// TIA Portal V19 export
FUNCTION_BLOCK "DelayOnOff"   // FB113, LAD
TITLE = Delay ON-OFF for sensor / DELAY ON/OFF
// stored: MemoryReserve 100, SetENOAutomatically false
   VAR_INPUT
      IN : Bool;
      DelayON : Time;
      DelayOFF : Time;
   END_VAR
   VAR_OUTPUT
      OUT : Bool;
   END_VAR
   VAR
      tonDelayOn : IEC_TIMER;
      tonDelayOff : IEC_TIMER;
   END_VAR
   VAR DB_SPECIFIC
      Result : Bool;
   END_VAR
BEGIN

REGION Network 1: Delay ON-OFF / Main
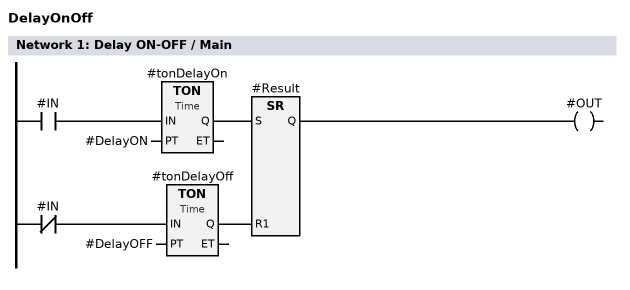
   RUNG wire#powerrail
      Contact( #IN )
      { S7_Templates := "time_type := Time" } #tonDelayOn.TON(pt := #DelayON, et =>)
      S_SR(operand := #Result, r1 := wire#w1)
      Coil( #OUT )
   END_RUNG
   RUNG wire#powerrail
      I_Contact( #IN )
      { S7_Templates := "time_type := Time" } #tonDelayOff.TON(pt := #DelayOFF, et =>)
   END_RUNG wire#w1
   // the same network as SCL:
   #tonDelayOn.TON(IN := #IN, PT := #DelayON);
   #tonDelayOff.TON(IN := NOT #IN, PT := #DelayOFF);
   IF #tonDelayOn.Q THEN
       #Result := TRUE;   // SR flip-flop
   END_IF;
   IF #tonDelayOff.Q THEN #Result := FALSE; END_IF;
   #OUT := #Result;
END_REGION
END_FUNCTION_BLOCK
